Staubli VAL3: Numerisation.pjx

--- Numerisation.pjx ---
Parameters version=s8.12.1cs9_BS2449 stackSize=200000 millimeterUnit=true
Program file=BalayageSimple.pgx
Program file=Communication.pgx
Program file=Deplacements.pgx
Program file=InitInterface.pgx
Program file=InitVariables.pgx
Program file=PositionUpdate.pgx
Program file=start.pgx
Program file=stop.pgx
Data file=Numerisation.dtx

--- Numerisation.dtx ---
bool bAcquisitionStarted = true
bool bOverrun
jointRx jCurrentJoint = {j1=-9.566067, j2=37.23348, j3=99.811939, j4=1.059303e-14, j5=42.95458, j6=-9.566067}
jointRx jCurrentJointError = {j1=0.00111051, j2=-0.000418031, j3=-0.000552065, j4=-0.00000679927, j5=-0.000103346, j6=0.000911689}
jointRx jInitialPosition = {j2=37.32, j3=99.65, j5=43.03}
jointRx jInitialPositionRepos = {j2=28.35, j3=97.17, j5=54.5}
jointRx jRobotZeroPosition = {j6=90}
mdesc mNomSpeed
num nBinaryPositionArray[24]
  [0] = 68
  [1] = 21
  [2] = 43
  [3] = 8
  [4] = 194
  [5] = 71
  [6] = 116
  [7] = 129
  [8] = 194
  [9] = 145
  [10] = 94
  [11] = 130
  [12] = 57
  [13] = 16
  [14] = 130
  [15] = 243
  [16] = 195
  [17] = 51
  [18] = 255
  [19] = 204
  [20] = 57
  [21] = 54
  [22] = 234
  [23] = 129
num nBinaryPositionArrayIndex
num nCurrentPositionArray[6]
  [0] = 596.672343
  [1] = -49.863772
  [2] = -72.684587
  [3] = 0.000137817
  [4] = -179.999203
  [5] = 0.000174442
num nMaxHorizontal = 1000
num nMaxRotation = 180
num nMaxVertical = 950
num nMinHorizontal = -1000
num nMinRotation = -180
num nMinVertical = -883.44
num nNextPositionX = 737.67
num nReceivedByte = 10
num nScanningLength = 200
num nScanningLineNumber = 5
num nScanningWidth = 200
pointRx pCircle = {x=497.67, y=50, z=-72.68, rx=-180, rz=-180, shoulder=sfree, elbow=efree, wrist=wfree, fatherId=world[0]}
pointRx pCurrentPosition = {x=596.760773, y=-49.877677, z=-72.686767, rx=0.000182979, ry=-179.998942, rz=0.000203803, shoulder=lefty, elbow=epositive, wrist=wpositive, fatherId=world[0]}
pointRx pInitialPosition = {x=597.67, y=50, z=-72.68, rx=-180, rz=-180, shoulder=sfree, elbow=efree, wrist=wfree, fatherId=world[0]}
pointRx pInitialPositionRepos = {x=597.67, y=50, z=27.32, rx=-180, rz=-180, shoulder=sfree, elbow=efree, wrist=wfree, fatherId=world[0]}
pointRx pNextPosition = {x=597.67, y=-50, z=-72.68, rx=-180, rz=-180, shoulder=sfree, elbow=efree, wrist=wfree, fatherId=world[0]}
pointRx pRobotZeroPosition = {x=50, y=50, z=950, shoulder=sfree, elbow=efree, wrist=wfree, fatherId=world[0]}
public sio sioSockets_c1 = {link=UdpSocket\c1}

--- start.pgx ---
program start()
begin
  call InitVariables()
  taskCreate "PositionUpdate",10,PositionUpdate()
  taskCreateSync "Communication",0.001,bOverrun,Communication()
  call InitInterface()
  call Deplacements()
end

--- BalayageSimple.pgx ---
program BalayageSimple()
begin
  //Rappel : pInitialPosition = {{597.67, 50, -72.68,-180,0,-180}, {sfree, efree, wfree}}
  while bAcquisitionStarted==false
  endWhile

  pNextPosition=pInitialPosition
  for nNextPositionX=pInitialPosition.trsf.x-nScanningLength/2 to pInitialPosition.trsf.x+nScanningLength/2 step nScanningLength/nScanningLineNumber
    pNextPosition.trsf.y=pInitialPosition.trsf.y-nScanningWidth/2
    pNextPosition.trsf.x=nNextPositionX
    movel(pNextPosition,flange,mNomSpeed)
    waitEndMove()
    pNextPosition.trsf.y=pInitialPosition.trsf.y+nScanningWidth/2
    movel(pNextPosition,flange,mNomSpeed)
    waitEndMove()
  endFor
  pNextPosition.trsf.x=pInitialPosition.trsf.x
  pNextPosition.trsf.y=pInitialPosition.trsf.y-nScanningWidth/2
  movec(pCircle,pNextPosition,flange,mNomSpeed)
  waitEndMove()
end

--- Communication.pgx ---
program Communication()
begin
  while true
    // Attente d'une demande d'acquisition (0xFE = 254). Quand on reçoit la demande, on attend une demande de position (0x01 = 1) ou de fin d'acquisition (0xEF = 239).
    nReceivedByte=sioSockets_c1
    if nReceivedByte==254
      // Demande d'acquisition reçu on commence
      bAcquisitionStarted=true

      while bAcquisitionStarted==true
        nReceivedByte=sioSockets_c1
        if nReceivedByte==1
          // Demande de position, on envoie pCurrentPosition
          nCurrentPositionArray[0]=pCurrentPosition.trsf.x
          nCurrentPositionArray[1]=pCurrentPosition.trsf.y
          nCurrentPositionArray[2]=pCurrentPosition.trsf.z
          nCurrentPositionArray[3]=pCurrentPosition.trsf.rx
          nCurrentPositionArray[4]=pCurrentPosition.trsf.ry
          nCurrentPositionArray[5]=pCurrentPosition.trsf.rz

          // Passage en binaire
          toBinary(nCurrentPositionArray,6,"4.0b",nBinaryPositionArray)

          // Envoi (2 start bytes (0xFE 0x7F + message)
          sioSockets_c1=254
          sioSockets_c1=127
          //for nBinaryPositionArrayIndex = 0 to 23
          sioSet(sioSockets_c1,nBinaryPositionArray)
          //          endFor

        elseIf nReceivedByte==239
          // Demande de fin d'acquisition reçu. On ne repart pas pour un tour.
          bAcquisitionStarted=false
        endIf
      endWhile
    endIf
  endWhile
end

--- Deplacements.pgx ---
program Deplacements()
begin
  //Déplacement vers la position initiale du robot, sert uniquement lors des simulations
  movej(pRobotZeroPosition,flange,mNomSpeed)

  //Déplacement vers une position initiale de numérisation
  //movel(pInitialPosition, flange, mNomSpeed)
  //waitEndMove()

  while true
    //Décalage vers le haut
    movel(pInitialPositionRepos,flange,mNomSpeed)
    waitEndMove()

    //Execution d'un balayage de surface
    call BalayageSimple()
  endWhile
end

--- InitInterface.pgx ---
program InitInterface()
begin
  //Open Interface
  userPage("InterfaceRobot")

  //Position Labels Bindings
  userPageBind("InterfaceRobot","lblXValue","innerHTML",pCurrentPosition.trsf.x,1,"r")
  userPageBind("InterfaceRobot","lblYValue","innerHTML",pCurrentPosition.trsf.y,1,"r")
  userPageBind("InterfaceRobot","lblZValue","innerHTML",pCurrentPosition.trsf.z,1,"r")
  userPageBind("InterfaceRobot","lblRXValue","innerHTML",pCurrentPosition.trsf.rx,1,"r")
  userPageBind("InterfaceRobot","lblRYValue","innerHTML",pCurrentPosition.trsf.ry,1,"r")
  userPageBind("InterfaceRobot","lblRZValue","innerHTML",pCurrentPosition.trsf.rz,1,"r")

  //Position Error Labels Bindings
  userPageBind("InterfaceRobot","lblJ1_errValue","innerHTML",jCurrentJointError.j1,1,"r")
  userPageBind("InterfaceRobot","lblJ2_errValue","innerHTML",jCurrentJointError.j2,1,"r")
  userPageBind("InterfaceRobot","lblJ3_errValue","innerHTML",jCurrentJointError.j3,1,"r")
  userPageBind("InterfaceRobot","lblJ4_errValue","innerHTML",jCurrentJointError.j4,1,"r")
  userPageBind("InterfaceRobot","lblJ5_errValue","innerHTML",jCurrentJointError.j5,1,"r")
  userPageBind("InterfaceRobot","lblJ6_errValue","innerHTML",jCurrentJointError.j6,1,"r")

  //Range Number Gauge Bindings : Values
  userPageBind("InterfaceRobot","rngX","value",pCurrentPosition.trsf.x,1,"r")
  userPageBind("InterfaceRobot","rngY","value",pCurrentPosition.trsf.y,1,"r")
  userPageBind("InterfaceRobot","rngZ","value",pCurrentPosition.trsf.z,1,"r")
  userPageBind("InterfaceRobot","rngRX","value",pCurrentPosition.trsf.rx,1,"r")
  userPageBind("InterfaceRobot","rngRY","value",pCurrentPosition.trsf.ry,1,"r")
  userPageBind("InterfaceRobot","rngRZ","value",pCurrentPosition.trsf.rz,1,"r")

  //Range Number Gauge Bindings : Low Limits
  userPageBind("InterfaceRobot","rngX","min",nMinHorizontal,1,"r")
  userPageBind("InterfaceRobot","rngY","min",nMinHorizontal,1,"r")
  userPageBind("InterfaceRobot","rngZ","min",nMinVertical,1,"r")
  userPageBind("InterfaceRobot","rngRX","min",nMinRotation,1,"r")
  userPageBind("InterfaceRobot","rngRY","min",nMinRotation,1,"r")
  userPageBind("InterfaceRobot","rngRZ","min",nMinRotation,1,"r")

  //Range Number Gauge Bindings : High Limits
  userPageBind("InterfaceRobot","rngX","max",nMaxHorizontal,1,"r")
  userPageBind("InterfaceRobot","rngY","max",nMaxHorizontal,1,"r")
  userPageBind("InterfaceRobot","rngZ","max",nMaxVertical,1,"r")
  userPageBind("InterfaceRobot","rngRX","max",nMaxRotation,1,"r")
  userPageBind("InterfaceRobot","rngRY","max",nMaxRotation,1,"r")
  userPageBind("InterfaceRobot","rngRZ","max",nMaxRotation,1,"r")

end

--- InitVariables.pgx ---
program InitVariables()
begin
  bAcquisitionStarted=false
  nReceivedByte=0

  //Dimensions balayage simple
  nScanningLength=200
  nScanningWidth=200
  nScanningLineNumber=20

  //Limites Ref. Cartésien (utiles pour affichage interface graphique)
  nMinHorizontal=-1000
  nMaxHorizontal=1000
  nMinVertical=-883.44
  nMaxVertical=950
  nMinRotation=-180
  nMaxRotation=180


  //Position initiale du robot
  jRobotZeroPosition={0,0,0,0,0,90}
  pRobotZeroPosition={{50,50,950,0,0,0},{sfree,efree,wfree}}

  //Position initiale de numérisation
  jInitialPosition={0,37.32,99.65,0,43.03,0}
  pInitialPosition={{597.67,50,-72.68,-180,0,-180},{sfree,efree,wfree}}

  jInitialPositionRepos={0,28.35,97.17,0,54.5,0}
  pInitialPositionRepos={{597.67,50,27.32,-180,0,-180},{sfree,efree,wfree}}

  //Position intermédiaire du cercle
  pCircle=pInitialPosition
  pCircle.trsf.x=pCircle.trsf.x-nScanningLength/2
end

--- PositionUpdate.pgx ---
program PositionUpdate()
begin
  while true
    jCurrentJoint=herej()
    jCurrentJointError=getPositionErr()
    pCurrentPosition=jointToPoint(flange,world,jCurrentJoint-jCurrentJointError)
    //pCurrentPosition = here(flange, world)
    delay(0.01)
  endWhile
end
